// TIA Portal V19 export
DATA_BLOCK "DB_FlatnessCtrlRecords"   // DB77
{ S7_Optimized_Access := 'TRUE'; DB_Accessible_From_OPC_UA := 'FALSE' }
// stored: AutoNumber false, DBAccessibleFromOPCUA false, DBAccessibleFromWebserver false, MemoryReserve 100
   VAR RETAIN
      LeftRobot { ExternalWritable := 'False'} : Struct
         uiNumberOfRecods : UInt;
         FlatnessRecords : Array[0..200] of "stFlatnessCtrlRecord";
      END_STRUCT;
      RightRobot { ExternalWritable := 'False'} : Struct
         uiNumberOfRecods : UInt;
         FlatnessRecords : Array[0..200] of "stFlatnessCtrlRecord";
      END_STRUCT;
   END_VAR
BEGIN
END_DATA_BLOCK
